(* Logix 5000 project; controller cal1615 1756-L62 rev 16.20; software revision 16.05; part 78 of 78 *)

PROGRAM ZZZ
END_PROGRAM
